// TIA Portal V15.1 export
// export: Created 2026-01-09T13:45:14.1150278Z, ExportSetting WithDefaults, WithReadOnly, DisplayName Totally Integrated Automation Portal, DisplayVersion V15.1 Update 8, DisplayName TIA Portal Openness, DisplayVersion V15.1 Update 8, DisplayName STEP 7 Professional, DisplayVersion V15.1 Update 8, DisplayName WinCC Advanced, DisplayVersion V15.1 Update 8
DATA_BLOCK "PLC_BIT"   // DB9
{ S7_Optimized_Access := 'FALSE' }
VERSION : 0.1
// stored: AutoNumber true, CodeModifiedDate 2026-01-01T12:46:58.5268647Z, CompileDate 2026-01-01T12:47:15.7550826Z, CreationDate 2024-10-12T12:36:08.0193576Z, DBAccessibleFromOPCUA true, InterfaceModifiedDate 2026-01-01T12:46:58.5268647Z, IsConsistent true, IsKnowHowProtected false, IsOnlyStoredInLoadMemory false, IsPLCDB false, IsWriteProtectedInAS false, ModifiedDate 2026-01-01T12:46:58.5268647Z, ParameterModified 2026-01-01T12:46:58.5268647Z, StructureModified 2026-01-01T12:46:58.5268647Z
   VAR
      RUN : Bool;
      MAN : Bool;
      AUT : Bool;
      SIM : Bool;
      PAU : Bool;
      NTR_FU : Bool;
      PCH_FU : Bool;
      SKIP_FU : Bool;
      AGG1_FU : Bool;
      WAG1_FU : Bool;
      WAG1_EM : Bool;
      AGG2_FU : Bool;
      WAG2_FU : Bool;
      WAG2_EM : Bool;
      AGG3_FU : Bool;
      WAG3_FU : Bool;
      WAG3_EM : Bool;
      AGG4_FU : Bool;
      WAG4_FU : Bool;
      WAG4_EM : Bool;
      AGG5_FU : Bool;
      WAG5_FU : Bool;
      WAG5_EM : Bool;
      AGG6_FU : Bool;
      WAG6_FU : Bool;
      WAG6_EM : Bool;
      CEM1_FU : Bool;
      CEM2_FU : Bool;
      CEM3_FU : Bool;
      WCE1_FU : Bool;
      WCE1_EM : Bool;
      CEM4_FU : Bool;
      CEM5_FU : Bool;
      WCE2_FU : Bool;
      WCE2_EM : Bool;
      WAT1_FU : Bool;
      WWA1_FU : Bool;
      WWA1_EM : Bool;
      WAT2_FU : Bool;
      WWA2_FU : Bool;
      WWA2_EM : Bool;
      ADD1_FU : Bool;
      ADD2_FU : Bool;
      ADD3_FU : Bool;
      WAD1_FU : Bool;
      WAD1_EM : Bool;
      ADD4_FU : Bool;
      ADD5_FU : Bool;
      ADD6_FU : Bool;
      WAD2_FU : Bool;
      WAD2_EM : Bool;
      "BAT/TAT NT" : Bool;
      "BAT/TAT BTX" : Bool;
      "NN_CAN NUOC" : Bool;
      "NN_XA NUOC" : Bool;
      NN_MCN : Bool;
      NN_DCN : Bool;
      "NN_DONG KEP" : Bool;
      "NN_MO KEP" : Bool;
      "NN_GAU LEN" : Bool;
      "NN_DUNG GAU" : Bool;
      "NN_GAU XUONG" : Bool;
      TOP_BTC : Bool;
      "TOP. GAU LEN" : Bool;
      "TOP. GAU XUONG" : Bool;
      "COT LIEU_FU" : Bool;
      PCĐ_SIM : Bool;
      PCM_SIM : Bool;
      CNĐ_SIM : Bool;
      CNM_SIM : Bool;
      "CN1/2_SIM" : Bool;
      COT_LIEU_FU : Bool;
      KT_XA_AGG : Bool;
      NEXT_WAGG1 : Bool;
      NEXT_WAGG2 : Bool;
      NEXT_WAGG3 : Bool;
      NEXT_WAGG4 : Bool;
      NEXT_WAGG5 : Bool;
      NEXT_WAGG6 : Bool;
      NEXT_WCEM1 : Bool;
      NEXT_WCEM2 : Bool;
      NEXT_WWAT1 : Bool;
      NEXT_WWAT2 : Bool;
      NEXT_WADD1 : Bool;
      NEXT_WADD2 : Bool;
      End_Agg1 : Bool;
      End_Agg2 : Bool;
      End_Agg3 : Bool;
      End_Agg4 : Bool;
      End_Agg5 : Bool;
      End_Agg6 : Bool;
      SW_MODE : Bool;
   END_VAR
BEGIN
END_DATA_BLOCK
